Staubli VAL3: numericalTwins.dtx

mdesc mNomSpeed
sio sioSocket = {link=Socket\test}
jointRx jHere
string sData
num nFrameIndex
num nEol
string sTaskPos
bool bOvrPosition
num nOvrPos
num nPrevOvrPos
string sTaskRobot
jointRx jStart
pointRx pPick = {fatherId=world[0]}
trsf trAppro
pointRx pPlace = {fatherId=world[0]}
